// TIA Portal V20 export
FUNCTION_BLOCK "FB_Digital_Outputs"   // FB3, LAD
{ S7_Optimized_Access := 'TRUE' }
// stored: AutoNumber false, MemoryReserve 100, SetENOAutomatically false
   VAR_INPUT
      DB_Blink_Button_Light : Bool;
      DB_Turn_On_Button_Light : Bool;
      DB_Light_Fail_Test : Bool;
      DB_Light_Approve_Test : Bool;
      DB_Digital_Output_3 : Bool;
      Clock_1Hz : Bool;
   END_VAR
   VAR_OUTPUT
      Q_Button_Light : Bool;
      Q_Light_Fail_Test : Bool;
      Q_Light_Approve_Test : Bool;
      Q_Digital_Output_3 : Bool;
   END_VAR
   VAR
      Timer_Delay_Fail_Test { S7_SetPoint := 'True'} : TON_TIME;
      Timer_Delay_Approve_Test { S7_SetPoint := 'True'} : TON_TIME;
   END_VAR
BEGIN

REGION Network 1
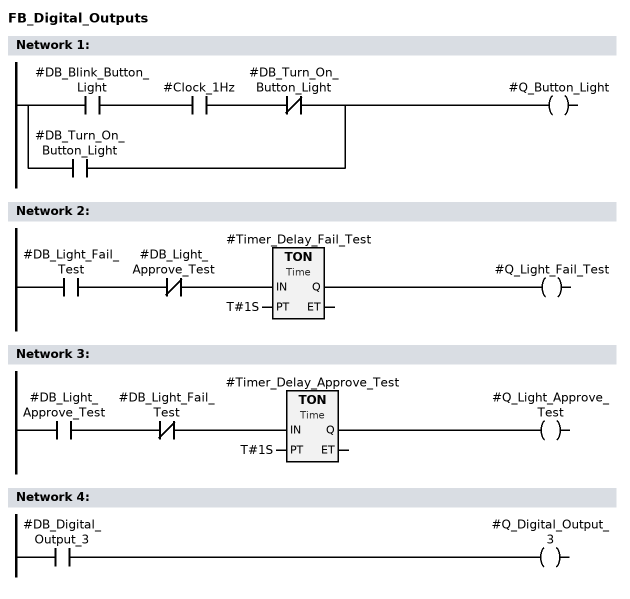
   RUNG wire#powerrail
      Contact( #DB_Blink_Button_Light )
      Contact( #Clock_1Hz )
      I_Contact( #DB_Turn_On_Button_Light )
      wire#w1
      Coil( #Q_Button_Light )
   END_RUNG
   RUNG wire#powerrail
      Contact( #DB_Turn_On_Button_Light )
   END_RUNG wire#w1
   // the same network as SCL:
   #Q_Button_Light := (#DB_Blink_Button_Light AND #Clock_1Hz AND NOT #DB_Turn_On_Button_Light) OR #DB_Turn_On_Button_Light;
END_REGION

REGION Network 2
   RUNG wire#powerrail
      Contact( #DB_Light_Fail_Test )
      I_Contact( #DB_Light_Approve_Test )
      { S7_Templates := "time_type := Time" } #Timer_Delay_Fail_Test.TON(pt := T#1S, et =>)
      Coil( #Q_Light_Fail_Test )
   END_RUNG
   // the same network as SCL:
   #Timer_Delay_Fail_Test(IN := #DB_Light_Fail_Test AND NOT #DB_Light_Approve_Test, PT := T#1S);   // TON
   #Q_Light_Fail_Test := #Timer_Delay_Fail_Test.Q;
END_REGION

REGION Network 3
   RUNG wire#powerrail
      Contact( #DB_Light_Approve_Test )
      I_Contact( #DB_Light_Fail_Test )
      { S7_Templates := "time_type := Time" } #Timer_Delay_Approve_Test.TON(pt := T#1S, et =>)
      Coil( #Q_Light_Approve_Test )
   END_RUNG
   // the same network as SCL:
   #Timer_Delay_Approve_Test(IN := #DB_Light_Approve_Test AND NOT #DB_Light_Fail_Test, PT := T#1S);   // TON
   #Q_Light_Approve_Test := #Timer_Delay_Approve_Test.Q;
END_REGION

REGION Network 4
   RUNG wire#powerrail
      Contact( #DB_Digital_Output_3 )
      Coil( #Q_Digital_Output_3 )
   END_RUNG
   // the same network as SCL:
   #Q_Digital_Output_3 := #DB_Digital_Output_3;
END_REGION
END_FUNCTION_BLOCK
